// TwinCAT 3 PLC project Modbus
// ProgramVersion: 3.1.4023.0
// libraries:
//   Tc2_ModbusSrv, * (Beckhoff Automation GmbH)
//   Tc2_Standard, * (Beckhoff Automation GmbH)
//   Tc2_System, * (Beckhoff Automation GmbH)
//   Tc3_Module, * (Beckhoff Automation GmbH)
//   VisuSymbols,3.5.10.0,System
// project tree:
//   / GlobalTextList.TcGTLO, Modbus_task.TcTTO, PlcTask.TcTTO, VisualizationManager.TcVMO (not stored)
//   GVLs/ GVL.TcGVL
//   POUs/ MAIN.TcPOU, pc.TcPOU, U_Convert.TcPOU
//   VISUs/ Visualization.TcVIS
// real-time tasks:
//   TASK PlcTask: cycle T#10ms, priority 20, ADS port 350
//   TASK Modbus_task: cycle T#10ms, priority 21, ADS port 351
//   TASK VISU_TASK: cycle T#200000us, priority 30, ADS port 352

CONFIGURATION Modbus
    RESOURCE PLC ON TwinCAT3
        TASK Modbus_task(INTERVAL := T#10ms, PRIORITY := 21);
        TASK PlcTask(INTERVAL := T#10ms, PRIORITY := 20);
        PROGRAM pc WITH Modbus_task : pc;
        PROGRAM MAIN WITH PlcTask : MAIN;
    END_RESOURCE
END_CONFIGURATION

// ---- GVLs/GVL.TcGVL
{attribute 'qualified_only'}
VAR_GLOBAL
	
fRealValue : REAL;

END_VAR

// ---- POUs/pc.TcPOU
PROGRAM pc
VAR
	cnt: INT;
	

 	//modbus
	MBReadRegs	: FB_MBReadRegs;
	fRealValude : REAL;
	MBReadArray	: ARRAY [0..4*4-1] OF BYTE;
	MBExecute	: BOOL;
	
	uConvert	: U_Convert;
	MB_i		: INT;
	MBRegs	 	: ARRAY [0..4-1] OF REAL;
	
END_VAR

cnt := cnt + 1;	

IF cnt >= 100 THEN
	cnt := 0;
END_IF

IF cnt <= 50 THEN	MBExecute := 1;	
ELSE 				MBExecute := 0;	
END_IF

MBReadRegs(
	sIPAddr:= '192.168.0.10',
	nTCPPort:= 504,
	nUnitID:= 16#FF,  
	nQuantity:= 2*4, 
	nMBAddr:= 0, 
	cbLength:= SIZEOF(MBReadArray), 
	pDestAddr:= ADR(MBReadArray),  
	bExecute:= MBExecute, 
	tTimeout:= T#1S, 
	bBusy=> , 
	bError=> , 
	nErrId=> , 
	cbRead=> ,
);

FOR MB_i:=1 TO 4 BY 1 DO
	//BYTE t o REAL
	uConvert.arrUDP_Data[0] := MBReadArray[2+4*MB_i-4]; // LSB
	uConvert.arrUDP_Data[1] := MBReadArray[3+4*MB_i-4];
	uConvert.arrUDP_Data[2] := MBReadArray[0+4*MB_i-4];
	uConvert.arrUDP_Data[3] := MBReadArray[1+4*MB_i-4]; // MSB
	MBRegs[MB_i-1] := uConvert.rReal;
END_FOR;

END_PROGRAM

// ---- POUs/U_Convert.TcPOU
TYPE U_Convert :  
	UNION  
		arrUDP_Data: ARRAY [0 .. 3] OF BYTE; // Array must start with LSB  
		rReal : REAL;  
	END_UNION  
END_TYPE

// ---- POUs/MAIN.TcPOU
PROGRAM MAIN
VAR
	cnt: INT;
	

 	//modbus
	MBReadRegs	: FB_MBReadRegs;
	fRealValude : REAL;
	MBReadArray	: ARRAY [0..4*4-1] OF BYTE;
	MBExecute	: BOOL;
	
	uConvert	: U_Convert;
	MB_i		: INT;
	MBRegs	 	: ARRAY [0..4-1] OF REAL;
	

END_VAR

cnt := cnt + 1;	

IF cnt >= 100 THEN
	cnt := 0;
END_IF

IF cnt <= 50 THEN	MBExecute := 1;	
ELSE 				MBExecute := 0;	
END_IF

MBReadRegs(
	sIPAddr:= '192.168.0.10',
	nTCPPort:= 504,
	nUnitID:= 16#FF,  
	nQuantity:= 2*4, 
	nMBAddr:= 0, 
	cbLength:= SIZEOF(MBReadArray), 
	pDestAddr:= ADR(MBReadArray),  
	bExecute:= MBExecute, 
	tTimeout:= T#1S, 
	bBusy=> , 
	bError=> , 
	nErrId=> , 
	cbRead=> ,
);

FOR MB_i:=1 TO 4 BY 1 DO
	//BYTE t o REAL
	uConvert.arrUDP_Data[0] := MBReadArray[2+4*MB_i-4]; // LSB
	uConvert.arrUDP_Data[1] := MBReadArray[3+4*MB_i-4];
	uConvert.arrUDP_Data[2] := MBReadArray[0+4*MB_i-4];
	uConvert.arrUDP_Data[3] := MBReadArray[1+4*MB_i-4]; // MSB
	MBRegs[MB_i-1] := uConvert.rReal;
END_FOR;

END_PROGRAM

// ---- VISUs/Visualization.TcVIS
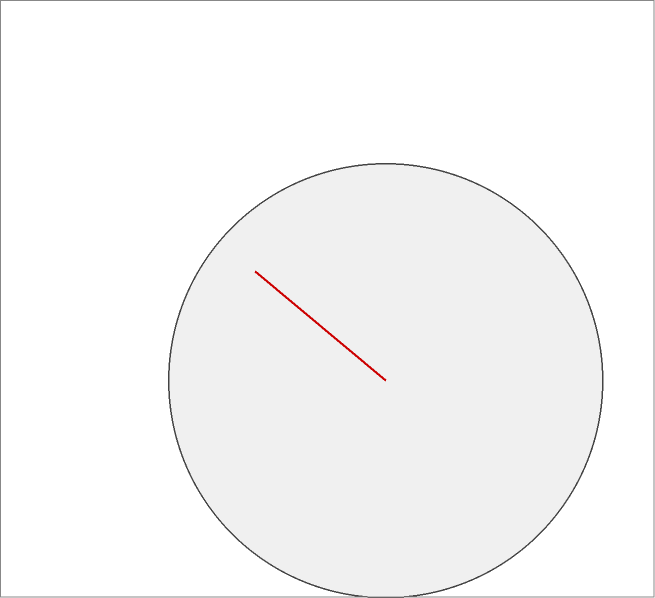
VISUALIZATION Visualization  // 655x598
    Meter180 (116,163 539x435), value: pc.MBRegs[0], style: Meter-Meter180-Gray, scale format: %.1f, scale 0..900
END_VISUALIZATION
